// TIA Portal V20 export
VAR_GLOBAL   // PLC tag table "Tag table_1"
END_VAR
